{attribute 'GeneratedUsingTerminal: AT2050-0500-0016'}
{attribute addProperty BoxType "AT2050-0500-0016"}
{attribute addProperty Id "EtcSlaveTerminalBaseCC_InputsAT %I*CC_Inputs_2C1C9EE032CC_OutputsAT %Q*CC_Outputs_69F9BE1432WcStateAT %I*WcState_9091E0EB2InfoDataAT %I*InfoData_BEF6B88E18"}
{attribute addProperty CRC "2249677633"}
{attribute addProperty Size "84"}
TYPE AT2050_86175B41 EXTENDS EtcSlaveTerminalBase :
STRUCT
	{attribute addProperty Name "CC_Inputs"}
	CC_Inputs : CC_Inputs_2C1C9EE0;
	{attribute addProperty Name "CC_Outputs"}
	CC_Outputs : CC_Outputs_69F9BE14;
	{attribute addProperty Name "WcState"}
	WcState : WcState_9091E0EB;
	{attribute addProperty Name "InfoData"}
	InfoData : InfoData_BEF6B88E;
END_STRUCT
END_TYPE

(* stored: Version 1.2.0.0, ProductVersion 3.1.4024.9
   DUT AT2050_86175B41: Id {b7d73312-6b54-4dc8-97ff-89069514b2c6} *)
